// TIA Portal V20 export
DATA_BLOCK "ProdDataInterfaceHmi"   // DB53
TITLE = HMI and user interface for production data
AUTHOR : SICAR
FAMILY : ProdData
// DESCRIPTION OF FUNCTIONS:
// stored: MemoryReserve 100
   VAR RETAIN
      numberOfDataSets : "LSicar_typeNumberOfDataSets";   // Number of configured data sets
   END_VAR
   VAR
      colorCodeLimitSummary : UInt;   // Overall status Limit values
      colorCodeLimitSelButton : Array[0..8] of UInt;   // Color code for data set select button (Limit values)
   END_VAR
   VAR RETAIN
      limitValueDataSetSel : Int := 1;   // selected data set limit values
      limitDataSet : Array[0.."NO_DATASETS_LIMITVALUES"] of "LSicar_typeLimitValue";   // Data sets limit .values
      cycleTimerDataSetSel : Int := 1;   // selected data set cycle timer
      cycleTimerDataSet : Array[0.."NO_DATASETS_CYCLETIMER"] of "LSicar_typeCycleTimer";   // Data sets cycle timer
      counterDataSetSel : Int := 1;   // selected data set counter
      counterDataSet : Array[0.."NO_DATASETS_COUNTER"] of "LSicar_typeCounter";   // Data sets counter
      shiftCounterDataSetSel : Int := 1;   // selected data set shift counter
      shiftCounterDataSet : Array[0.."NO_DATASETS_SHIFTCOUNTER"] of "LSicar_typeShiftCounter";   // Data sets shift counter
      shiftCountOeeDataSetSel : Int := 1;   // selected data set OEE
      shiftCounterOeeDataSet : Array[0.."NO_DATASETS_SHIFTCOUNTER"] of "LSicar_typeShiftCounterOee";   // Data sets shift counter OEE
   END_VAR
BEGIN
END_DATA_BLOCK
